Yaskawa INFORM job: R1_W53-A2(90,90).JBI

/JOB
//NAME R1_W53-A2(90,90)
///FOLDERNAME KRIS-SCIANA
//POS
///NPOS 54,54,0,2,0,0
///TOOL 0
///POSTYPE PULSE
///PULSE
C00000=125464,54795,11916,11,80425,-11658
C00001=121260,36987,11214,6722,73303,-26770
C00002=121230,46639,38017,7289,61852,-27463
C00003=122241,53153,48068,7083,58944,-27260
C00004=122994,55656,52047,6863,57731,-27040
C00005=122980,57562,54200,6894,57389,-27067
C00006=122635,56026,52462,7013,57691,-27185
C00007=115735,75335,76366,23767,62426,-33932
C00008=116402,75107,76087,23601,62287,-33691
C00009=115735,75335,76366,23767,62426,-33932
C00010=122958,70240,66479,6151,63242,-27072
C00011=122958,71102,68653,6199,62352,-27121
C00012=122949,71417,67723,6164,63083,-27086
C00013=122579,68264,62659,6197,64599,-27143
C00014=121633,61461,51491,6314,68030,-27307
C00015=120725,86942,86965,-6360,96130,703
C00016=120725,94594,101296,-6306,91272,948
C00017=120866,95828,104140,-6267,90169,1047
C00018=120720,91828,98455,-6309,91597,931
C00019=120722,104658,115687,-6298,87608,1131
C00020=120725,96386,105145,-6300,89833,1018
C00021=120725,94590,101320,-6306,91255,949
C00022=120725,86929,86977,-6360,96117,703
C00023=120724,66094,58037,-4026,59743,-41882
C00024=120724,68322,64308,-4142,57035,-41781
C00025=120775,56844,55427,-4471,51144,-41516
C00026=120602,68569,64801,-4100,56853,-41823
C00027=120553,66518,62749,-4070,57059,-41850
C00028=122230,56905,55497,-5227,51220,-40897
C00029=120724,67441,61892,-5047,61541,-36174
C00030=120724,65441,55931,-4933,64172,-36290
C00031=120500,45149,7307,-4433,83593,-37110
C00032=145452,77818,44713,-11922,79884,-28597
C00033=156803,-4554,-21296,-38868,71085,-35796
C00034=145388,-53117,-46253,-49880,51520,-42437
C00035=153251,-10376,-12137,-57408,89787,-31071
C00036=152418,-12344,-11713,-57378,88572,-30739
C00037=155236,19602,15444,-62294,108365,-24509
C00038=153863,24819,24400,-61587,106099,-23539
C00039=146924,20502,28447,-59274,98703,-22584
C00040=144263,18847,29999,-58387,95867,-22218
C00041=141947,-406,14710,-60739,85177,-25031
C00042=141719,1448,17330,-60050,86083,-17288
C00043=141210,-455,15065,-60828,84595,-25059
C00044=141032,770,15718,-60833,84600,-25181
C00045=140006,424,16470,-60248,85030,-17586
C00046=141965,-1146,16183,-62420,84073,-23333
C00047=144263,18847,29999,-58387,95867,-22218
C00048=147702,19244,24221,-58394,100004,-23066
C00049=152047,-13313,-8676,-60691,86268,-28928
C00050=145388,-53117,-46253,-49880,51520,-42437
C00051=145388,-54648,-53588,-47775,54028,-44022
C00052=145387,-55124,-68255,-43768,60279,-47394
C00053=70536,-76246,-94484,-49862,51525,-42441
BC00000=79590,530020,1075173
BC00001=74772,511583,1075175
BC00002=74772,511583,1075175
BC00003=74772,511583,1075175
BC00004=74772,511583,1075171
BC00005=74772,511583,1075171
BC00006=74772,511583,1075175
BC00007=74772,511583,1075175
BC00008=74772,511583,1075175
BC00009=74772,511583,1075175
BC00010=74772,511583,1075175
BC00011=74772,511583,1075175
BC00012=74772,511583,1075175
BC00013=74772,511583,1075175
BC00014=74772,511583,1075175
BC00015=38069,470864,1075175
BC00016=38985,470210,1075175
BC00017=39227,470058,1075174
BC00018=39352,469948,1075175
BC00019=39352,469948,1075175
BC00020=46883,469938,1075175
BC00021=46517,470200,1075175
BC00022=45600,470854,1075175
BC00023=55686,520112,1075175
BC00024=53159,516957,1075175
BC00025=52148,515695,1075175
BC00026=52148,515695,1075175
BC00027=52148,515695,1075175
BC00028=52148,515695,1075175
BC00029=47332,512764,1075175
BC00030=49711,516085,1075175
BC00031=49711,516085,1075175
BC00032=49711,516085,1075175
BC00033=17908,450192,1075175
BC00034=15,413119,1075175
BC00035=15,413119,1075175
BC00036=15,413119,1075175
BC00037=15,413119,1075175
BC00038=15,413119,1075175
BC00039=15,413119,1075175
BC00040=15,413119,1075175
BC00041=15,413620,1075175
BC00042=15,413300,1075172
BC00043=15,412678,1075175
BC00044=15,412678,1075175
BC00045=15,413300,1075172
BC00046=15,413300,1075172
BC00047=15,413119,1075175
BC00048=15,413119,1075175
BC00049=15,413119,1075175
BC00050=15,413119,1075175
BC00051=15,413119,1075175
BC00052=76033,557880,1075171
BC00053=76033,593253,1075171
///POSTYPE BASE
///RECTAN
///RCONF 0,0,0,0,1,0,0,0,0,0,0,0,0,0,0,0,0,0,0,0,0,0,0,0
P00006=2.006,1.622,-0.565,0.0000,0.0000,0.0000
P00022=2.006,1.622,-0.565,0.0000,0.0000,0.0000
//INST
///DATE 2025/06/06 11:53
///ATTR SC,RW
///GROUP1 RB1,BS1
NOP
'Path S980
SFTOF
MOVJ C00000 BC00000 VJ=100.00
MOVJ C00001 BC00001 VJ=100.00
MOVJ C00002 BC00002 VJ=20.00
MOVL C00003 BC00003 V=100.0
MOVL C00004 BC00004 V=60.0
REFP 3 C00005 BC00005
CALL JOB:SEARCH-R1
SET P022 P006
SFTON P022
MOVL C00006 BC00006 V=60.0
MOVL C00007 BC00007 V=60.0
REFP 3 C00008 BC00008
CALL JOB:SEARCH-R1
SET P022 P006
SFTON P022
MOVL C00009 BC00009 V=60.0
MOVL C00010 BC00010 V=60.0
REFP 3 C00011 BC00011
CALL JOB:SEARCH-R1
SET P022 P006
SFTON P022
MOVL C00012 BC00012 V=60.0
MOVL C00013 BC00013 V=100.0
MOVL C00014 BC00014 V=100.0
'Path W981
SFTOF
SFTON P022
MOVL C00015 BC00015 V=100.0
MOVL C00016 BC00016 V=100.0
MOVL C00017 BC00017 V=100.0 PL=0
REFP 1 C00018 BC00018
REFP 2 C00019 BC00019
MACRO1 MJ#(0) ARGF7
ARCON
MOVL C00020 BC00020 V=10.0
ARCOF
MOVL C00021 BC00021 V=100.0
MOVL C00022 BC00022 V=100.0
SFTOF
'Path W982
SFTOF
SFTON P022
MOVJ C00023 BC00023 VJ=20.00
MOVL C00024 BC00024 V=100.0
MOVL C00025 BC00025 V=100.0 PL=0
REFP 1 C00026 BC00026
REFP 2 C00027 BC00027
MACRO1 MJ#(0) ARGF7
ARCON
MOVL C00028 BC00028 V=8.3
ARCOF
MOVL C00029 BC00029 V=100.0
MOVL C00030 BC00030 V=16.7
SFTOF
'Path VIA1071
SFTOF
MOVJ C00031 BC00031 VJ=20.00
'Path VIA1072
SFTOF
MOVJ C00032 BC00032 VJ=20.00
MOVJ C00033 BC00033 VJ=20.00
MOVJ C00034 BC00034 VJ=20.00
SFTOF
MOVJ C00035 BC00035 VJ=10.00
MOVJ C00036 BC00036 VJ=20.00
MOVJ C00037 BC00037 VJ=10.00
MOVJ C00038 BC00038 VJ=15.00
'Path VIA1069
SFTOF
'Path VIA1067
SFTOF
MOVJ C00039 BC00039 VJ=15.00
MOVJ C00040 BC00040 VJ=10.00
'Path W983
SFTOF
SFTON P022
MOVL C00041 BC00041 V=100.0
MOVL C00042 BC00042 V=100.0 PL=0
REFP 1 C00043 BC00043
REFP 2 C00044 BC00044
MACRO1 MJ#(0) ARGF7
ARCON
MOVL C00045 BC00045 V=10.0
ARCOF
MOVL C00046 BC00046 V=100.0
SFTOF
'Path VIA1063
SFTOF
MOVJ C00047 BC00047 VJ=10.00
'Path VIA1064
SFTOF
MOVJ C00048 BC00048 VJ=10.00
'Path VIA1065
SFTOF
MOVJ C00049 BC00049 VJ=10.00
'Path VIA1066
SFTOF
MOVJ C00050 BC00050 VJ=20.00
MOVJ C00051 BC00051 VJ=100.00
'COMMENT
MOVJ C00052 BC00052 VJ=100.00
MOVJ C00053 BC00053 VJ=100.00
END
